FUNCTION_BLOCK ControlPLCcomp (* Composite Function Block Type *)
  (* Standard: 61499-2 *)
  (* Version 0.0, 7/26/2023, vv263, nxtControl GmBH, template *)
  PACKAGE Main;
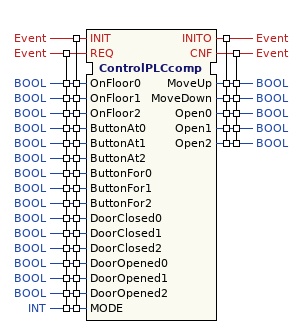
  EVENT_INPUT
    INIT WITH OnFloor0, OnFloor1, OnFloor2, ButtonAt0, ButtonAt1, ButtonAt2, ButtonFor0, ButtonFor1, ButtonFor2, DoorClosed0, DoorClosed1, DoorClosed2, DoorOpened0, DoorOpened1, DoorOpened2, MODE;
    REQ WITH OnFloor0, OnFloor1, OnFloor2, ButtonAt0, ButtonAt1, ButtonAt2, ButtonFor0, ButtonFor1, ButtonFor2, DoorClosed0, DoorClosed1, DoorClosed2, DoorOpened0, DoorOpened1, DoorOpened2, MODE;
  END_EVENT
  EVENT_OUTPUT
    INITO WITH MoveUp, MoveDown, Open0, Open1, Open2;
    CNF WITH MoveUp, MoveDown, Open0, Open1, Open2;
  END_EVENT
  VAR_INPUT
    OnFloor0 : BOOL; (* Input event qualifier *)
    OnFloor1 : BOOL;
    OnFloor2 : BOOL;
    ButtonAt0 : BOOL;
    ButtonAt1 : BOOL;
    ButtonAt2 : BOOL;
    ButtonFor0 : BOOL;
    ButtonFor1 : BOOL;
    ButtonFor2 : BOOL;
    DoorClosed0 : BOOL;
    DoorClosed1 : BOOL;
    DoorClosed2 : BOOL;
    DoorOpened0 : BOOL;
    DoorOpened1 : BOOL;
    DoorOpened2 : BOOL;
    MODE : INT := 1;
  END_VAR
  VAR_OUTPUT
    MoveUp : BOOL; (* Output event qualifier *)
    MoveDown : BOOL;
    Open0 : BOOL;
    Open1 : BOOL;
    Open2 : BOOL;
  END_VAR
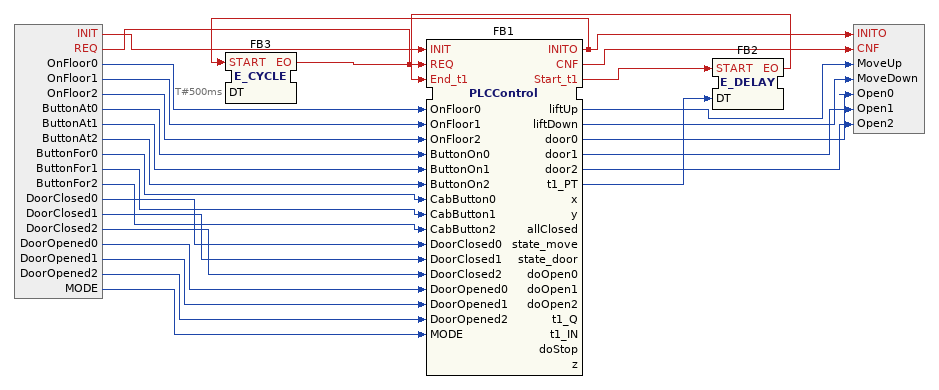
  FBS
    FB1 : PLCControl;
    FB2 : E_DELAY;
    FB3 : E_CYCLE(DT := T#500ms);
  END_FBS
  EVENT_CONNECTIONS
    FB1.INITO TO INITO;
    FB1.CNF TO CNF;
    INIT TO FB1.INIT;
    FB1.Start_t1 TO FB2.START;
    FB2.EO TO FB1.End_t1;
    FB1.INITO TO FB3.START;
    FB3.EO TO FB1.REQ;
    REQ TO FB1.REQ;
  END_CONNECTIONS
  DATA_CONNECTIONS
    OnFloor0 TO FB1.OnFloor0;
    OnFloor1 TO FB1.OnFloor1;
    OnFloor2 TO FB1.OnFloor2;
    DoorClosed0 TO FB1.DoorClosed0;
    DoorClosed1 TO FB1.DoorClosed1;
    DoorClosed2 TO FB1.DoorClosed2;
    ButtonAt0 TO FB1.ButtonOn0;
    ButtonAt1 TO FB1.ButtonOn1;
    ButtonAt2 TO FB1.ButtonOn2;
    ButtonFor0 TO FB1.CabButton0;
    ButtonFor1 TO FB1.CabButton1;
    ButtonFor2 TO FB1.CabButton2;
    FB1.liftUp TO MoveUp;
    FB1.liftDown TO MoveDown;
    DoorOpened0 TO FB1.DoorOpened0;
    DoorOpened1 TO FB1.DoorOpened1;
    DoorOpened2 TO FB1.DoorOpened2;
    FB1.door0 TO Open0;
    FB1.door1 TO Open1;
    FB1.door2 TO Open2;
    FB1.t1_PT TO FB2.DT;
    MODE TO FB1.MODE;
  END_CONNECTIONS
END_FUNCTION_BLOCK
